Staubli VAL3: page_viewTraj.dtx

num nIndex
num nKey = 255
num nOldIndex = 2
public num nPage
num nRefresh = 13186.401
num nSelect
num nTime = 0.1
num nView
num nClockStatus
string sEvent = " 3. "
public string sItems = "test"
string sList[3]
  [0] = " 1. "
  [1] = " 2. "
  [2] = " 3. "
string sMenu[8]
  [0] = "Tool Selection"
  [2] = "Rename"
  [3] = "Paste"
  [4] = "Mark"
  [5] = "Delete"
  [6] = "Insert"
  [7] = "Save"
string sMenuUser[8]
string sMessage
string sTrajName = "test"
string sMenu8[8]
bool bButton[8]
  [0] = true
  [2] = true
  [3] = true
  [4] = true
  [5] = true
  [6] = true
  [7] = true
bool bLarge
bool bShowStatus
bool bExit
bool bTrigger
tool tTool = {fatherId=flange[0], ioLink=valve1}
frame fFather = {fatherId=world[0]}
num nBackupFrame
public string Stest[2]
string l_sltem
public string sWorkingmode[10]
  [0] = "1号石墨舟A面取片"
  [1] = "1号石墨舟A面放片"
  [2] = "1号石墨舟B面取片"
  [3] = "1号石墨舟B面放片"
  [4] = "2号石墨舟A面取片"
  [5] = "2号石墨舟A面放片"
  [6] = "2号石墨舟B面取片"
  [7] = "2号石墨舟B面放片"
  [8] = "花篮取片"
  [9] = "花篮放片"
num nSelected
